FUNCTION_BLOCK FB_Tempering
VAR_INPUT
	bExecute		: BOOL;
END_VAR
VAR_OUTPUT
	bDone			: BOOL;
	bError			: BOOL;
	wErrorID		: BOOL;
END_VAR
VAR
	
END_VAR

END_FUNCTION_BLOCK

(* stored: Version 1.1.0.1, ProductVersion 3.1.4024.11
   POU FB_Tempering: Id {c38b8cdc-1856-4303-be47-22d52c579c56}, SpecialFunc None *)
